PROGRAM DoSomeMath
VAR
	rValue1	: REAL	:= 7;	
	rValue2	: REAL	:= 2;
	rResult	: REAL	:= 0;
	
	iCounter : INT := 0;
	
	//Test Array
	aTestArray 	: ARRAY[0..10] OF INT;
	iTestValue	: INT := 0;
	
END_VAR

rResult := f_Addition(rSum1 := rValue1, rSum2 := rValue2);
rResult := f_Multiplication(rValue1, rValue2);
rResult := f_Division(aTestArray[2], rValue2);
iCounter := iCounter + 1;

FOR iTestValue := 0 TO 10 BY 1 DO
	aTestArray[iTestValue] := iCounter;
	 IF iTestValue >3 THEN
		 EXIT;
	 END_IF
END_FOR

END_PROGRAM

(* stored: Version 1.1.0.1, ProductVersion 3.1.4024.12
   POU DoSomeMath: Id {4a75e5f3-85b5-4cc5-abda-38066dc40cd2}, SpecialFunc None *)
